/// Rolling interval to create a new log file when expired. 
{attribute 'qualified_only'}
{attribute 'strict'}
{attrivute 'to_string'}
TYPE RollingIntervals :
(
	None := 0,
	Hourly,
	Daily,
	Monthly
);
END_TYPE

(* stored: Version 1.1.0.1
   DUT RollingIntervals: Id {6a02719a-974a-441f-b806-8e74fa123285} *)
